// TIA Portal project "Project2" (V15)

(* hardware
DEVICE "HMI_1"  TP1200 Comfort
   slot 0: "HMI_1"  TP1200 Comfort  6AV2 124-0MC01-0AX0  15.0.0.0
   slot 1: "HMI_RT_1"  TP1200 Comfort  6AV2 124-0MC01-0AX0  15.0.0.0
   slot 5: "HMI_1.IE_CP_1"  PROFINET Interface  15.0.0.0
      slot 1: "PROFINET Interface_1"  PROFINET Interface
         slot 1: "Port_1"  Port
         slot 2: "Port_2"  Port
   slot 7: "HMI_1.MPI/DP_CP_1"  MPI/DP Interface  15.0.0.0
*)

(* ===== HMI "HMI_RT_1" =====
system functions are stored by id; their names below are inferred from use
connection "Connection_1": OPC, OPC_UA

HMI tags "Default tag table"
   "Tag_ScreenNumber" : Int, internal

HMI tags "Rpi3WiFi"
   "WiFi1_SSID" : String[14] AT ns=http://opcfoundation.org/RpiWiFiOpcUa;i=15099, 5 s
   "WiFi2_SSID" : String[14] AT ns=http://opcfoundation.org/RpiWiFiOpcUa;i=15100, 5 s
   "WiFi3_SSID" : String[14] AT ns=http://opcfoundation.org/RpiWiFiOpcUa;i=15101, 5 s
   "WiFi4_SSID" : String[14] AT ns=http://opcfoundation.org/RpiWiFiOpcUa;i=15102, 5 s
   "WiFi5_SSID" : String[14] AT ns=http://opcfoundation.org/RpiWiFiOpcUa;i=15103, 5 s
   "WiFi_PassKey" : String[100] AT ns=http://opcfoundation.org/RpiWiFiOpcUa;i=15104, 5 s
   "WiFi1_IsConnected" : Boolean AT ns=http://opcfoundation.org/RpiWiFiOpcUa;i=15105, 5 s
   "WiFi2_IsConnected" : Boolean AT ns=http://opcfoundation.org/RpiWiFiOpcUa;i=15106, 5 s
   "WiFi3_IsConnected" : Boolean AT ns=http://opcfoundation.org/RpiWiFiOpcUa;i=15107, 5 s
   "WiFi4_IsConnected" : Boolean AT ns=http://opcfoundation.org/RpiWiFiOpcUa;i=15108, 5 s
   "WiFi5_IsConnected" : Boolean AT ns=http://opcfoundation.org/RpiWiFiOpcUa;i=15109, 5 s
   "WiFi1_ConnectCmd" : Boolean AT ns=http://opcfoundation.org/RpiWiFiOpcUa;i=15110, 5 s
   "WiFi2_ConnectCmd" : Boolean AT ns=http://opcfoundation.org/RpiWiFiOpcUa;i=15111, 5 s
   "WiFi3_ConnectCmd" : Boolean AT ns=http://opcfoundation.org/RpiWiFiOpcUa;i=15112, 5 s
   "WiFi4_ConnectCmd" : Boolean AT ns=http://opcfoundation.org/RpiWiFiOpcUa;i=15113, 5 s
   "WiFi5_ConnectCmd" : Boolean AT ns=http://opcfoundation.org/RpiWiFiOpcUa;i=15114, 5 s
   "WiFi_DisconnectCmd" : Boolean AT ns=http://opcfoundation.org/RpiWiFiOpcUa;i=15117, 5 s
   "WiFi6_ConnectCmd" : Boolean AT ns=http://opcfoundation.org/RpiWiFiOpcUa;i=15077, 5 s
   "WiFi6_IsConnected" : Boolean AT ns=http://opcfoundation.org/RpiWiFiOpcUa;i=15072, 5 s
   "WiFi6_SSID" : String[14] AT ns=http://opcfoundation.org/RpiWiFiOpcUa;i=15066, 5 s
   "WiFi7_ConnectCmd" : Boolean AT ns=http://opcfoundation.org/RpiWiFiOpcUa;i=15078, 5 s
   "WiFi7_IsConnected" : Boolean AT ns=http://opcfoundation.org/RpiWiFiOpcUa;i=15073, 5 s
   "WiFi7_SSID" : String[14] AT ns=http://opcfoundation.org/RpiWiFiOpcUa;i=15067, 5 s
   "WiFi8_ConnectCmd" : Boolean AT ns=http://opcfoundation.org/RpiWiFiOpcUa;i=15079, 5 s
   "WiFi8_IsConnected" : Boolean AT ns=http://opcfoundation.org/RpiWiFiOpcUa;i=15074, 5 s
   "WiFi8_SSID" : String[14] AT ns=http://opcfoundation.org/RpiWiFiOpcUa;i=15068, 5 s
   "WiFi9_ConnectCmd" : Boolean AT ns=http://opcfoundation.org/RpiWiFiOpcUa;i=15080, 5 s
   "WiFi9_IsConnected" : Boolean AT ns=http://opcfoundation.org/RpiWiFiOpcUa;i=15075, 5 s
   "WiFi9_SSID" : String[14] AT ns=http://opcfoundation.org/RpiWiFiOpcUa;i=15070, 5 s
   "WiFi10_ConnectCmd" : Boolean AT ns=http://opcfoundation.org/RpiWiFiOpcUa;i=15081, 5 s
   "WiFi10_IsConnected" : Boolean AT ns=http://opcfoundation.org/RpiWiFiOpcUa;i=15076, 5 s
   "WiFi10_SSID" : String[14] AT ns=http://opcfoundation.org/RpiWiFiOpcUa;i=15071, 5 s

screen "Root screen" 1280x740, template "Template_1"
   on GenerateScreen: SetTag("Tag_ScreenNumber", 1)
   TextField "Text field_1" at 163,101 size 17x25; Text '1'
   TextField "Text field_2" at 163,146 size 17x25; Text '2'
   TextField "Text field_3" at 163,191 size 17x25; Text '3'
   TextField "Text field_4" at 163,236 size 17x25; Text '4'
   TextField "Text field_5" at 163,282 size 17x25; Text '5'
   IOField "I/O field_1" at 207,95 size 437x32; FormatPattern ??????????????
      ProcessValue <- "WiFi1_SSID"
   IOField "I/O field_2" at 207,140 size 437x32; FormatPattern ??????????????
      ProcessValue <- "WiFi2_SSID"
   IOField "I/O field_3" at 207,186 size 437x32; FormatPattern ??????????????
      ProcessValue <- "WiFi3_SSID"
   IOField "I/O field_4" at 207,231 size 437x32; FormatPattern ??????????????
      ProcessValue <- "WiFi4_SSID"
   IOField "I/O field_5" at 207,277 size 437x32; FormatPattern ??????????????
      ProcessValue <- "WiFi5_SSID"
   Button "Button_1" at 794,91 size 192x38; TextOff 'Connect to 1'
      on Click: SetBit("WiFi1_ConnectCmd")
   IOField "I/O field_6" at 704,16 size 351x32; FormatPattern ??????????????????????????????
      ProcessValue <- "WiFi_PassKey"
   TextField "Text field_6" at 571,19 size 128x25; Text 'WiFi Passkey'
   Button "Button_2" at 794,136 size 192x38; TextOff 'Connect to 2'
      on Click: SetBit("WiFi2_ConnectCmd")
   Button "Button_3" at 794,182 size 192x38; TextOff 'Connect to 3'
      on Click: SetBit("WiFi3_ConnectCmd")
   Button "Button_4" at 794,227 size 192x38; TextOff 'Connect to 4'
      on Click: SetBit("WiFi4_ConnectCmd")
   Button "Button_5" at 794,273 size 192x38; TextOff 'Connect to 5'
      on Click: SetBit("WiFi5_ConnectCmd")
   TextField "Text field_7" at 673,52 size 105x25; Text 'Connected'
   TextField "Text field_8" at 252,53 size 99x25; Text 'WiFi SSID'
   Circle "Circle_1" at 702,94 size 31x31
      Appearance <- "WiFi1_IsConnected"
   Circle "Circle_2" at 702,139 size 31x31
      Appearance <- "WiFi2_IsConnected"
   Circle "Circle_3" at 702,276 size 31x31
      Appearance <- "WiFi5_IsConnected"
   Circle "Circle_4" at 702,230 size 31x31
      Appearance <- "WiFi4_IsConnected"
   Circle "Circle_5" at 702,185 size 31x31
      Appearance <- "WiFi3_IsConnected"
   Button "Button_6" at 1074,17 size 192x38; TextOff 'Disconnect WiFi'
      on Click: SetBit("WiFi_DisconnectCmd")
   TextField "Text field_9" at 163,330 size 17x25; Text '6'
   TextField "Text field_10" at 163,375 size 17x25; Text '7'
   TextField "Text field_11" at 163,420 size 17x25; Text '8'
   TextField "Text field_12" at 163,465 size 17x25; Text '9'
   TextField "Text field_13" at 163,511 size 29x25; Text '10'
   IOField "I/O field_7" at 207,324 size 437x32; FormatPattern ??????????????
      ProcessValue <- "WiFi6_SSID"
   IOField "I/O field_8" at 207,369 size 437x32; FormatPattern ??????????????
      ProcessValue <- "WiFi7_SSID"
   IOField "I/O field_9" at 207,415 size 437x32; FormatPattern ??????????????
      ProcessValue <- "WiFi8_SSID"
   IOField "I/O field_10" at 207,460 size 437x32; FormatPattern ??????????????
      ProcessValue <- "WiFi9_SSID"
   IOField "I/O field_11" at 207,506 size 437x32; FormatPattern ??????????????
      ProcessValue <- "WiFi10_SSID"
   Button "Button_7" at 794,320 size 192x38; TextOff 'Connect to 6'
      on Click: SetBit("WiFi6_ConnectCmd")
   Button "Button_8" at 794,365 size 192x38; TextOff 'Connect to 7'
      on Click: SetBit("WiFi7_ConnectCmd")
   Button "Button_9" at 794,411 size 192x38; TextOff 'Connect to 8'
      on Click: SetBit("WiFi8_ConnectCmd")
   Button "Button_10" at 794,456 size 192x38; TextOff 'Connect to 9'
      on Click: SetBit("WiFi9_ConnectCmd")
   Button "Button_11" at 794,502 size 192x38; TextOff 'Connect to 10'
      on Click: SetBit("WiFi10_ConnectCmd")
   Circle "Circle_6" at 702,323 size 31x31
      Appearance <- "WiFi6_IsConnected"
   Circle "Circle_7" at 702,368 size 31x31
      Appearance <- "WiFi7_IsConnected"
   Circle "Circle_8" at 702,505 size 31x31
      Appearance <- "WiFi10_IsConnected"
   Circle "Circle_9" at 702,459 size 31x31
      Appearance <- "WiFi9_IsConnected"
   Circle "Circle_10" at 702,414 size 31x31
      Appearance <- "WiFi8_IsConnected"

Template "Template_1" 1280x740
   Button "Exit" at 1200,679 size 78x59; TextOff 'Exit'; PictureOff "ExitRuntime_TP1200_Comfort_TR"; PictureOn "ExitRuntime_TP1200_Comfort_TR"
      on Release: StopRuntime(0)
   Button "Template_Button" at 1120,679 size 78x59; TextOff 'Text'
   Button "Template_Button_1" at 1040,679 size 78x59; TextOff 'Text'
   Button "Template_Button_2" at 960,679 size 78x59; TextOff 'Text'
   Button "Template_Button_3" at 880,679 size 78x59; TextOff 'Text'
   Button "Template_Button_4" at 800,679 size 78x59; TextOff 'Text'
   Button "Template_Button_5" at 720,679 size 78x59; TextOff 'Text'
   Button "Template_Button_6" at 640,679 size 78x59; TextOff 'Text'
   Button "Template_Button_7" at 561,679 size 78x59; TextOff 'Text'
   Button "Template_Button_8" at 481,679 size 78x59; TextOff 'Text'
   Button "Template_Button_9" at 401,679 size 78x59; TextOff 'Text'
   Button "Template_Button_10" at 321,679 size 78x59; TextOff 'Text'
   Button "Template_Button_11" at 241,679 size 78x59; TextOff 'Text'
   Button "Template_Button_12" at 161,679 size 78x59; TextOff 'Text'
   Button "Template_Button_13" at 81,679 size 78x59; TextOff 'Text'
   Button "Start screen" at 1,679 size 78x59; TextOff 'Start screen'; PictureOff "NavigateHome_TP1200_Comfort_TR"; PictureOn "NavigateHome_TP1200_Comfort_TR"
      on Release: ActivateScreen("Root screen", 0)
*)